FUNCTION_BLOCK valve_analog
VAR_INPUT
	//Position Feedback from Valve
	position_feedback : REAL; 
	//Position Request from PLC Program
	position_request : REAL;
	//True when valve does not reach position in time
	fault : BOOL;
	// Position deadband for fail to reach position alarm
	position_deadband_sp: REAL;
	//Position valve should move to when faulted
	position_faulted : REAL;
END_VAR
VAR_OUTPUT
	//Position Command to Device
	position_command : REAL;
	// Position Deadband High for fail to reach position alarm
	position_deadband_high: REAL;
	// Position Deadband Low for fail to reach position alarm
	position_deadband_low: REAL;
	// Valve status, 0=Closed, 1=Open, 2=Middle, 3=Faulted
	status: INT;
END_VAR
VAR	
	// Position deadband, calculated value for fail to reach position alarm
	position_deadband: REAL;
	// If position feedback is less than this value, valve status will show closed.
	status_closed_percent: INT :=2;
	// If position feedback is greater than this value, valve status will show open
	status_open_percent : INT :=98;
END_VAR
VAR // added by the converter: edge detectors and wires of the graphical bodies
    _w1, _w2, _w3, _w4, _w5, _w6 : BOOL;
END_VAR

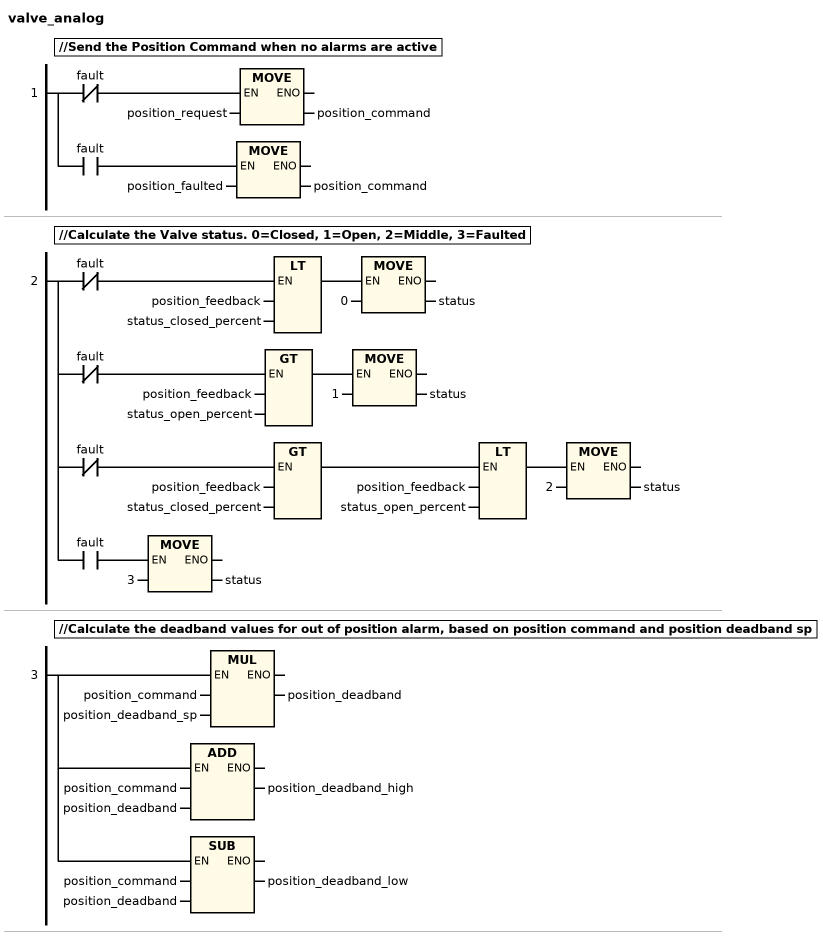
// NETWORK 1
// label: //Send the Position Command when no alarms are active
_w1 := NOT fault;
IF _w1 THEN position_command := position_request; END_IF
_w2 := fault;
IF _w2 THEN position_command := position_faulted; END_IF

// NETWORK 2
// label: //Calculate the Valve status. 0=Closed, 1=Open, 2=Middle, 3=Faulted
_w3 := NOT fault AND position_feedback < status_closed_percent;
IF _w3 THEN status := 0; END_IF
_w4 := NOT fault AND position_feedback > status_open_percent;
IF _w4 THEN status := 1; END_IF
_w5 := NOT fault AND position_feedback > status_closed_percent AND position_feedback < status_open_percent;
IF _w5 THEN status := 2; END_IF
_w6 := fault;
IF _w6 THEN status := 3; END_IF

// NETWORK 3
// label: //Calculate the deadband values for out of position alarm, based on position command and position deadband sp
position_deadband := position_command * position_deadband_sp;
position_deadband_high := position_command + position_deadband;
position_deadband_low := position_command - position_deadband;

END_FUNCTION_BLOCK

(* stored: Version 1.1.0.1, ProductVersion 3.1.4024.12
   POU valve_analog: Id {eb81a680-634a-469e-846c-a6f21734bdb6}, SpecialFunc None *)
